// TIA Portal V20 export
TYPE "LER_typeCommunicationSpecialFunctionsReelCut"
// stored: Access Published
   STRUCT
      specialFunction1 : Bool;
      specialFunction2 : Bool;
      specialFunction3 : Bool;
      specialFunction4 : Bool;
      specialFunction5 : Bool;
      specialFunction6 : Bool;
      specialFunction7 : Bool;
      specialFunction8 : Bool;
      specialFunction9 : Bool;
      specialFunction10 : Bool;
      specialFunction11 : Bool;
      specialFunction12 : Bool;
      specialFunction13 : Bool;
      specialFunction14 : Bool;
      specialFunction15 : Bool;
      specialFunction16 : Bool;
      specialFunction17 : Bool;
      specialFunction18 : Bool;
      specialFunction19 : Bool;
      specialFunction20 : Bool;
      specialFunction21 : Bool;
      specialFunction22 : Bool;
      specialFunction23 : Bool;
      specialFunction24 : Bool;
      specialFunction25 : Bool;
      specialFunction26 : Bool;
      specialFunction27 : Bool;
      specialFunction28 : Bool;
      specialFunction29 : Bool;
      specialFunction30 : Bool;
      specialFunction31 : Bool;
      specialFunction32 : Bool;
      specialFunction33 : Bool;
      specialFunction34 : Bool;
      specialFunction35 : Bool;
      specialFunction36 : Bool;
      specialFunction37 : Bool;
      specialFunction38 : Bool;
      specialFunction39 : Bool;
      specialFunction40 : Bool;
      specialFunction41 : Bool;
      specialFunction42 : Bool;
      specialFunction43 : Bool;
      specialFunction44 : Bool;
      specialFunction45 : Bool;
      specialFunction46 : Bool;
      specialFunction47 : Bool;
      specialFunction48 : Bool;
      specialFunction49 : Bool;
      specialFunction50 : Bool;
      specialFunction51 : Bool;
      specialFunction52 : Bool;
      specialFunction53 : Bool;
      specialFunction54 : Bool;
      specialFunction55 : Bool;
      specialFunction56 : Bool;
      specialFunction57 : Bool;
      specialFunction58 : Bool;
      specialFunction59 : Bool;
      specialFunction60 : Bool;
      specialFunction61 : Bool;
      specialFunction62 : Bool;
      specialFunction63 : Bool;
      specialFunction64 : Bool;
   END_STRUCT;
END_TYPE
